TYPE ST_VisionProcessConfig :
STRUCT
    eMode : E_VisionMode;
    tDetectionDelay : TIME;
    // Simulation模式下的原始检测角度，仅用于监控和诊断。
    fSimulatedDetectedAngle : LREAL;
    // Simulation模式下已经完成坐标及方向映射的DamperRotation修正量。
    fSimulatedCorrectionAngle : LREAL;
    bSimulatedDetected : BOOL;
    fSimulatedConfidence : LREAL;
    // 单次DamperRotation修正死区；不是二次视觉质量复检容差。
    fAngleTolerance : LREAL;
END_STRUCT
END_TYPE

(* stored: Version 1.1.0.1, ProductVersion 3.1.4026.20
   DUT ST_VisionProcessConfig: Id {42274acc-75c3-4a04-812c-ebbc4875d172} *)
